// TIA Portal V20 export
TYPE "UDT_Interlock_Flejadora"
   STRUCT
      Bit_0_Tipo_Flejado : Bool;
      Bit_1_Tipo_Flejado : Bool;
      Inicio_Flejado : Bool;
      Transportador_en_avance : Bool;
      "Byte0.bit4" : Bool;
      "Byte0.bit5" : Bool;
      "Byte0.bit6" : Bool;
      EMERGENCIA : Bool;
      Byte1_bit0 : Bool;
      Byte1_bit1 : Bool;
      Byte1_bit2 : Bool;
      Byte1_bit3 : Bool;
      Byte1_bit4 : Bool;
      Byte1_bit5 : Bool;
      Byte1_bit6 : Bool;
      Byte1_bit7 : Bool;
      Fin_Flejado : Bool;
      Flejadora_Operativa : Bool;
      Bypass_Flejadora : Bool;
      Move_OK_Flejadora : Bool;
      Byte2_bit4 : Bool;
      Byte2_bit5 : Bool;
      Byte2_bit6 : Bool;
      Byte2_bit7 : Bool;
      Byte3_bit0 : Bool;
      Byte3_bit1 : Bool;
      Byte3_bit2 : Bool;
      Byte3_bit3 : Bool;
      Byte3_bit4 : Bool;
      Byte3_bit5 : Bool;
      Byte3_bit6 : Bool;
      Byte3_bit7 : Bool;
   END_STRUCT;
END_TYPE
